Staubli VAL3: sendPacket.pgx

program sendPacket(num& x_nBuff[], num x_nSize)
  local num l_nIndex
begin

  resize(nTempBuffer,1,1)
  nTempBuffer=0
  if x_nSize>0
    resize(nTempBuffer,1,x_nSize)
  else
    call setLastError(nErrTCPSend)
    return
  endIf

  for l_nIndex=0 to x_nSize-1
    nTempBuffer[l_nIndex]=x_nBuff[l_nIndex]
  endFor

  //if the server is down this function is blocking this:
  //if watch(sioSet(sTCPclient, nTempBuffer) == size(nTempBuffer), nRecvTimeout)
  //...doesnt work because sioSet is blocked!...maybe we need to do this in a separate task and wait a response from this task!

  if sioSet(sTCPclient, nTempBuffer) != size(nTempBuffer)
    call setLastError(nErrTCPConnRst)
  endIf

end
